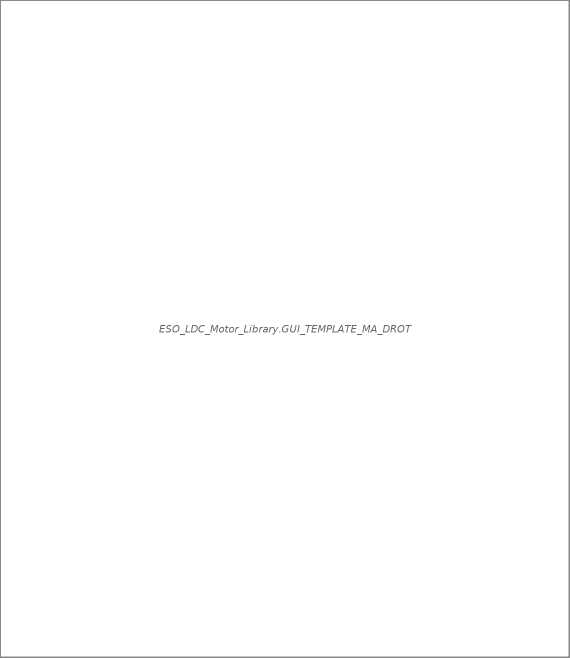
VISUALIZATION GUI_Drot  // 570x658
    Frame (0,0 570x658)
        shows ESO_LDC_Motor_Library.GUI_TEMPLATE_MA_DROT(m_DeviceName := 'drot', m_Instance := MAIN.drot)
END_VISUALIZATION

(* stored: Version 1.1.0.1, ProductVersion 3.1.4024.11
   Visu GUI_Drot: Id {68084031-ade7-460f-aad8-d91f25d0c50f} *)
